FUNCTION_BLOCK FB_Car EXTENDS FB_Vehicle

VAR
END_VAR

METHOD Model
VAR_INPUT
END_VAR
sOutput:= 'MODEL Number is :  CAMN0035E021004';
END_METHOD

END_FUNCTION_BLOCK

(* stored: Version 1.1.0.1, ProductVersion 3.1.4024.16
   POU FB_Car: Id {f8002561-94b2-4079-8a8d-200c7815a106}, SpecialFunc None
   Method Model: Id {9676e5b3-5d40-4db0-a6c9-ba694e34ee10} *)
